PROGRAM POU11
VAR
END_VAR

END_PROGRAM

(* stored: Version 1.1.0.1, ProductVersion 3.1.4024.6
   POU POU11: Id {72f8079d-9744-4eaf-b09b-d0f4d955c356}, SpecialFunc None *)
